FUNCTION_BLOCK ModbusTCPClient (* Template for a simple Basic Function Block Type *)
  (* Standard: 61499-2; Function: Modbus TCP Client; Description: Modbus TCP Client which connects to a Modbus device. The registers are made available to the applicaton *)
  (* Version 1.0, 2024-07-21, david *)
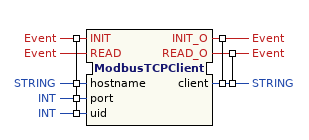
  EVENT_INPUT
    INIT WITH hostname, port, uid; (* Initialization Request *)
    READ; (* Normal Execution Request *)
  END_EVENT
  EVENT_OUTPUT
    INIT_O WITH client; (* Initialization Confirm *)
    READ_O WITH client; (* Execution Confirmation *)
  END_EVENT
  VAR_INPUT
    hostname : STRING; (* Hostname or IP of Modbus Device *)
    port : INT := 502; (* Port of Modbus Device *)
    uid : INT := 71; (* unit id *)
  END_VAR
  VAR_OUTPUT
    client : STRING; (* client Object *)
  END_VAR
END_FUNCTION_BLOCK
